// Mitsubishi GX Works2 project: LAB1.2   PLC: FX1N/FX1NC

PROGRAM MAIN
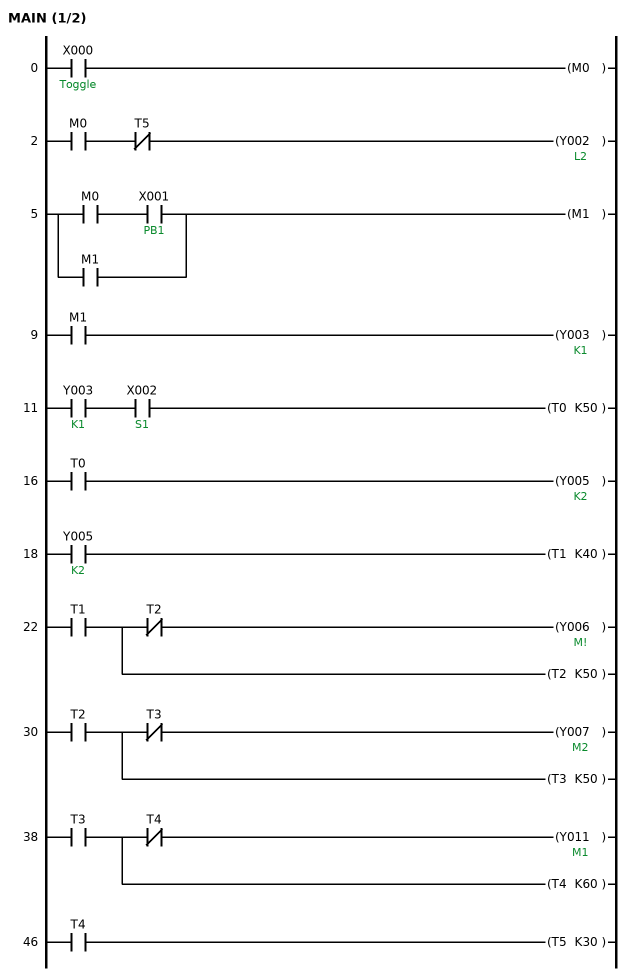
0     LD      X000  ; Toggle
      OUT     M0
2     LD      M0
      ANI     T5
      OUT     Y002  ; L2
5     LD      M0
      AND     X001  ; PB1
      OR      M1
      OUT     M1
9     LD      M1
      OUT     Y003  ; K1
11    LD      Y003  ; K1
      AND     X002  ; S1
      OUT     T0 K50
16    LD      T0
      OUT     Y005  ; K2
18    LD      Y005  ; K2
      OUT     T1 K40
22    LD      T1
      MPS
      ANI     T2
      OUT     Y006  ; M!
      MPP
      OUT     T2 K50
30    LD      T2
      MPS
      ANI     T3
      OUT     Y007  ; M2
      MPP
      OUT     T3 K50
38    LD      T3
      MPS
      ANI     T4
      OUT     Y011  ; M1
      MPP
      OUT     T4 K60
46    LD      T4
      OUT     T5 K30
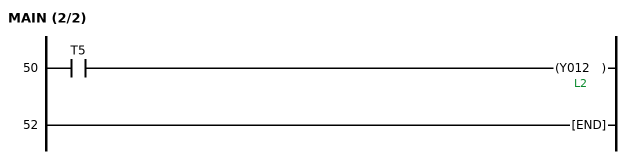
50    LD      T5
      OUT     Y012  ; L2
52    END
END_PROGRAM

// device comments not shown above
Y004  ; S1
